INTERFACE I_HaveNodes

END_INTERFACE

(* stored: Version 1.1.0.1, ProductVersion 3.1.4024.12
   Itf I_HaveNodes: Id {8b00edd2-48ce-0038-1549-5f98651536cb} *)
